TEXTLIST CRAH_Isolator_Status
  0 = 'OFF'
  1 = 'ON'
   = ''
END_TEXTLIST

(* stored: Version 1.1.0.1, ProductVersion 3.1.4024.12
   TextList CRAH_Isolator_Status: Id {99082a96-ab60-4b64-a689-507fed9c376f} *)
